FUNCTION_BLOCK FB_SLIDER (* A slider input *)
  (* Standard: 61499-1; ApplicationDomain: GUI; Function: Slider input *)
  (* Version 0.3, 2008-06-04, JHC, Holobloc Inc, Updated DOCTYPE. *)
  (* Version 0.2, 2001-03-04, JHC, Rockwell Automation, Udated documentation. *)
  (* Version 0.1, 2000-04-27, JHC, Rockwell Automation, Corrected IVAL handling. *)
  (* Compiler header: package fb.rt.hmi; import java.awt.*; import java.awt.event.*; *)
  (* Compiler Java IBM VisualAge 3.0 *)
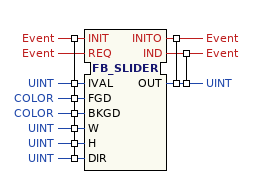
  EVENT_INPUT
    INIT WITH IVAL, FGD, BKGD, W, H, DIR; (* Initialization Request *)
    REQ; (* Read the current value *)
  END_EVENT
  EVENT_OUTPUT
    INITO WITH OUT; (* Initialization Confirm *)
    IND WITH OUT; (* REQ Confirmation or change of state *)
  END_EVENT
  VAR_INPUT
    IVAL : UINT; (* Initial slider position *)
    FGD : COLOR := red; (* Foreground Color *)
    BKGD : COLOR := blue; (* Background Color *)
    W : UINT := 75; (* Bar width *)
    H : UINT := 20; (* Bar height *)
    DIR : UINT; (* Orientation:0=L/R,1=T/B,2=R/L,3=B/T *)
  END_VAR
  VAR_OUTPUT
    OUT : UINT; (* Slider position{0..100} *)
  END_VAR
  SERVICE FB_SLIDER/component
    SEQUENCE initialization
      FB_SLIDER.INIT(IVAL,FGD,BKGD,W,H,DIR) -> component.init() -> FB_SLIDER.INITO(OUT);
    END_SEQUENCE
    SEQUENCE read_value
      FB_SLIDER.REQ() -> component.getValue() -> FB_SLIDER.CNF(OUT);
    END_SEQUENCE
    SEQUENCE update
      component.mouseEvent() -> FB_SLIDER.IND(OUT);
    END_SEQUENCE
  END_SERVICE
END_FUNCTION_BLOCK
